Yaskawa INFORM job: OK_R2_O49(180,90)AWOK.JBI

/JOB
//NAME OK_R2_O49(180,90)AWOK
///FOLDERNAME X4
//POS
///NPOS 112,112,112,7,0,0
///TOOL 0
///POSTYPE PULSE
///PULSE
C00000=-57370,-49169,-35389,-92398,112235,2416
C00001=-57338,-39846,-12309,-87938,111954,7208
C00002=-61668,-40068,-12639,-88811,108884,7066
C00003=-63399,-40053,-12708,-89154,107656,7009
C00004=-65644,-43123,-14595,-89423,106041,7176
C00005=-66050,-42449,-14221,-89539,105759,7114
C00006=-65644,-43123,-14595,-89423,106041,7176
C00007=-63399,-40053,-12708,-89154,107656,7009
C00008=-65860,-35872,-10226,-89816,105931,6667
C00009=-67308,-37830,-11473,-89989,104891,6764
C00010=-65860,-35872,-10226,-89816,105931,6667
C00011=-63399,-40053,-12708,-89154,107656,7009
C00012=-61668,-40068,-12639,-88811,108884,7066
C00013=-57338,-39846,-12309,-87938,111954,7208
C00014=-57370,-49169,-35389,-92398,112235,2416
C00015=-56766,-48274,-34752,-92403,112675,2380
C00016=-56734,-38983,-11654,-87839,112385,7203
C00017=-61035,-39257,-12018,-88706,109335,7062
C00018=-61363,-41475,-13444,-88660,109088,7185
C00019=-65079,-42508,-14107,-89322,106443,7178
C00020=-65354,-42062,-13862,-89401,106251,7134
C00021=-65079,-42508,-14107,-89322,106443,7178
C00022=-62757,-39264,-12100,-89046,108114,7005
C00023=-65205,-35368,-10154,-89778,106406,6571
C00024=-66729,-37471,-11499,-89953,105309,6677
C00025=-65205,-35368,-10154,-89778,106406,6571
C00026=-62757,-39264,-12100,-89046,108114,7005
C00027=-61035,-39257,-12018,-88706,109335,7062
C00028=-56734,-38983,-11654,-87839,112385,7203
C00029=-56766,-48274,-34752,-92403,112675,2380
C00030=-56218,-47521,-34536,-92505,113073,2248
C00031=-56187,-38348,-11498,-87842,112791,7100
C00032=-59131,-40673,-13118,-88322,110687,7128
C00033=-64463,-43713,-15068,-89195,106879,7202
C00034=-65258,-42417,-14335,-89420,106324,7084
C00035=-65041,-42755,-14501,-89355,106475,7122
C00036=-62171,-38696,-11986,-89025,108542,6906
C00037=-64564,-34510,-9127,-89599,106856,6674
C00038=-65923,-36436,-10368,-89757,105878,6764
C00039=-64564,-34510,-9127,-89599,106856,6674
C00040=-62171,-38696,-11986,-89025,108542,6906
C00041=-60460,-38670,-11893,-88691,109758,6961
C00042=-56187,-38348,-11498,-87842,112791,7100
C00043=-58012,-44746,-32893,-92770,111760,2043
C00044=-165233,-62484,-24672,90805,98196,-8817
C00045=-158022,-60427,-23957,92500,93160,-8513
C00046=-156743,-62313,-24995,92752,92269,-8672
C00047=-155558,-59411,-23565,93051,91431,-8394
C00048=-156743,-62313,-24995,92752,92269,-8672
C00049=-159918,-59160,-23326,92117,94487,-8388
C00050=-157669,-55497,-21549,92669,92903,-8023
C00051=-156702,-56139,-21884,92856,92223,-8084
C00052=-158315,-55054,-21316,92545,93357,-7983
C00053=-165233,-62484,-24672,90805,98196,-8817
C00054=-166433,-62392,-24374,90502,99029,-8891
C00055=-159182,-60473,-23727,92230,93972,-8588
C00056=-156333,-62291,-24667,92831,91984,-8760
C00057=-155539,-60352,-23718,93033,91424,-8573
C00058=-155684,-62672,-24851,92972,91532,-8802
C00059=-160153,-59816,-23401,92033,94651,-8523
C00060=-157527,-54468,-21504,92741,92796,-7792
C00061=-156419,-55217,-21907,92950,92016,-7861
C00062=-158582,-53729,-21112,92546,93541,-7724
C00063=-166433,-62392,-24374,90502,99029,-8891
C00064=-167171,-61612,-24215,90395,99552,-8755
C00065=-159973,-59772,-23597,92089,94525,-8457
C00066=-156562,-61998,-24743,92795,92141,-8668
C00067=-155803,-60186,-23919,92988,91604,-8474
C00068=-156562,-61998,-24743,92795,92141,-8668
C00069=-161445,-58729,-23074,91799,95557,-8358
C00070=-159459,-54024,-20839,92339,94160,-7872
C00071=-157637,-55308,-21529,92681,92878,-7984
C00072=-159252,-54174,-20918,92377,94014,-7885
C00073=-167171,-61612,-24215,90395,99552,-8755
C00074=-69409,-72138,-29447,-102463,36685,-80534
C00075=-71059,-73457,-30006,-103635,35630,-80116
C00076=-71839,-65365,-14695,-121986,41568,-74598
C00077=-70275,-72833,-29744,-103069,36130,-80318
C00078=-70612,-75418,-30749,-104190,36042,-79744
C00079=-72072,-56824,-1188,-125861,43468,-72277
C00080=-72838,-56347,-1048,-126291,42972,-72187
C00081=-73459,-46502,14196,-130452,45167,-69730
C00082=-73645,-58678,-6398,-124927,41399,-73193
C00083=-74008,-49012,8836,-129230,43689,-70644
C00084=-74555,-56613,-4486,-125720,40959,-72905
C00085=-74921,-46134,12069,-130385,43538,-70149
C00086=-75408,-55045,-3275,-126310,40460,-72728
C00087=-76023,-45250,12243,-130982,42784,-70051
C00088=-76728,-63195,-18080,-121997,37141,-75456
C00089=-77109,-54539,-3849,-127025,39193,-72649
C00090=-77504,-63710,-20410,-121159,36115,-76041
C00091=-77952,-55004,-5860,-126648,38177,-73027
C00092=-56542,-67334,-11423,-115165,51876,-75640
C00093=-67053,-69065,-28106,-99490,40183,15728
C00094=-67428,-69282,-26772,-100738,40056,16409
C00095=-67529,-60027,-12907,-115722,44463,22502
C00096=-65920,-70446,-28647,-99537,41009,15920
C00097=-68407,-70268,-28636,-100327,39293,16023
C00098=-67953,-51806,517,-119653,45920,24933
C00099=-68254,-60297,-14375,-115388,43715,22147
C00100=-68715,-51405,-117,-119604,45208,24719
C00101=-69350,-59817,-14851,-115483,42822,22008
C00102=-69870,-50869,-354,-119971,44342,24699
C00103=-70281,-60433,-17733,-114511,41681,21256
C00104=-70732,-50629,-1414,-119808,43487,24415
C00105=-71119,-50129,-1155,-119967,43215,24435
C00106=-71532,-39226,16503,-124978,45598,27505
C00107=-71875,-64574,-28650,-110190,39078,18480
C00108=-72245,-56839,-15158,-115347,40339,21445
C00109=-72519,-46657,1943,-121015,42457,24796
C00110=-72775,-36077,19150,-125892,44947,27780
C00111=-71161,-41775,15932,-125497,46306,27939
BC00000=398174,725769,70942
BC00001=398174,725769,70942
BC00002=398174,725769,70942
BC00003=398174,725769,70942
BC00004=398174,725769,70942
BC00005=398174,725769,70942
BC00006=398174,725769,70942
BC00007=398174,725769,70942
BC00008=398174,725769,70942
BC00009=398174,725769,70942
BC00010=398174,725769,70942
BC00011=398174,725769,70942
BC00012=398174,725769,70942
BC00013=398174,725769,70942
BC00014=398174,725769,70942
BC00015=398174,720870,420591
BC00016=398174,720870,420591
BC00017=398174,720870,420591
BC00018=398174,720870,420591
BC00019=398174,720870,420591
BC00020=398174,720870,420591
BC00021=398174,720870,420591
BC00022=398174,720870,420591
BC00023=398174,720870,420591
BC00024=398174,720870,420591
BC00025=398174,720870,420591
BC00026=398174,720870,420591
BC00027=398174,720870,420591
BC00028=398174,720870,420591
BC00029=398174,720870,420591
BC00030=398174,716148,751922
BC00031=398174,716148,751922
BC00032=398174,716148,751922
BC00033=398174,716148,751922
BC00034=398174,716148,751922
BC00035=398174,716148,751922
BC00036=398174,716148,751922
BC00037=398174,716148,751922
BC00038=398174,716148,751922
BC00039=398174,716148,751922
BC00040=398174,716148,751922
BC00041=398174,716148,751922
BC00042=398174,716148,751922
BC00043=398174,689571,751922
BC00044=15,723854,63219
BC00045=15,723854,63219
BC00046=15,723854,63219
BC00047=15,723854,63219
BC00048=15,723854,63219
BC00049=15,723854,63219
BC00050=15,723854,63219
BC00051=15,723854,63219
BC00052=15,723854,63219
BC00053=15,723854,63219
BC00054=15,720076,395244
BC00055=15,720076,395244
BC00056=15,720076,395244
BC00057=15,720076,395244
BC00058=15,720076,395244
BC00059=15,720076,395244
BC00060=15,720076,395244
BC00061=15,720076,395244
BC00062=15,720076,395244
BC00063=15,720076,395244
BC00064=15,714414,759792
BC00065=15,714414,759792
BC00066=15,714414,759792
BC00067=15,714414,759792
BC00068=15,714414,759792
BC00069=15,714414,759792
BC00070=15,714414,759792
BC00071=15,714414,759792
BC00072=15,714414,759792
BC00073=15,714414,759792
BC00074=15,669680,870811
BC00075=15,676887,869700
BC00076=15,679769,869255
BC00077=15,679769,869255
BC00078=15,679769,869255
BC00079=15,679769,869255
BC00080=15,679769,794529
BC00081=15,679769,794529
BC00082=15,679769,652674
BC00083=15,679769,652674
BC00084=15,679769,530552
BC00085=15,679769,530552
BC00086=15,679769,409308
BC00087=15,679769,409308
BC00088=15,679769,241527
BC00089=15,679769,241527
BC00090=15,679769,105258
BC00091=15,679769,105258
BC00092=15,679769,105258
BC00093=308901,670741,873357
BC00094=311453,677596,872312
BC00095=311410,677544,872261
BC00096=312666,680852,871816
BC00097=312666,680852,871816
BC00098=311410,677544,872261
BC00099=311409,677551,750069
BC00100=311409,677551,750069
BC00101=311409,677551,629774
BC00102=311409,677551,629774
BC00103=311409,677551,498785
BC00104=311409,677551,498785
BC00105=311409,677551,426569
BC00106=311409,677551,426569
BC00107=311409,677551,187001
BC00108=311409,677551,187001
BC00109=311409,677551,187001
BC00110=311409,677551,187001
BC00111=311409,677551,187001
EC00000=1596313,556475
EC00001=1596313,556475
EC00002=1596313,556475
EC00003=1596313,556475
EC00004=1596313,556475
EC00005=1596313,556475
EC00006=1596313,556475
EC00007=1596313,556475
EC00008=1596313,556475
EC00009=1596313,556475
EC00010=1596313,556475
EC00011=1596313,556475
EC00012=1596313,556475
EC00013=1596313,556475
EC00014=1596313,556475
EC00015=1596313,556475
EC00016=1596313,556475
EC00017=1596313,556475
EC00018=1596313,556475
EC00019=1596313,556475
EC00020=1596313,556475
EC00021=1596313,556475
EC00022=1596313,556475
EC00023=1596313,556475
EC00024=1596313,556475
EC00025=1596313,556475
EC00026=1596313,556475
EC00027=1596313,556475
EC00028=1596313,556475
EC00029=1596313,556475
EC00030=1596313,556475
EC00031=1596313,556475
EC00032=1596313,556475
EC00033=1596313,556475
EC00034=1596313,556475
EC00035=1596313,556475
EC00036=1596313,556475
EC00037=1596313,556475
EC00038=1596313,556475
EC00039=1596313,556475
EC00040=1596313,556475
EC00041=1596313,556475
EC00042=1596313,556475
EC00043=1596313,556475
EC00044=1596313,556475
EC00045=1596313,556475
EC00046=1596313,556475
EC00047=1596313,556475
EC00048=1596313,556475
EC00049=1596313,556475
EC00050=1596313,556475
EC00051=1596313,556475
EC00052=1596313,556475
EC00053=1596313,556475
EC00054=1596313,556475
EC00055=1596313,556475
EC00056=1596313,556475
EC00057=1596313,556475
EC00058=1596313,556475
EC00059=1596313,556475
EC00060=1596313,556475
EC00061=1596313,556475
EC00062=1596313,556475
EC00063=1596313,556475
EC00064=1596313,556475
EC00065=1596313,556475
EC00066=1596313,556475
EC00067=1596313,556475
EC00068=1596313,556475
EC00069=1596313,556475
EC00070=1596313,556475
EC00071=1596313,556475
EC00072=1596313,556475
EC00073=1596313,556475
EC00074=1596313,556475
EC00075=1596313,556475
EC00076=1596313,556475
EC00077=1596313,556475
EC00078=1596313,556475
EC00079=1596313,556475
EC00080=1596313,556475
EC00081=1596313,556475
EC00082=1596313,556475
EC00083=1596313,556475
EC00084=1596313,556475
EC00085=1596313,556475
EC00086=1596313,556475
EC00087=1596313,556475
EC00088=1596313,556475
EC00089=1596313,556475
EC00090=1596313,556475
EC00091=1596313,556475
EC00092=1596313,556475
EC00093=1596313,556475
EC00094=1596313,556475
EC00095=1596313,556475
EC00096=1596313,556475
EC00097=1596313,556475
EC00098=1596313,556475
EC00099=1596313,556475
EC00100=1596313,556475
EC00101=1596313,556475
EC00102=1596313,556475
EC00103=1596313,556475
EC00104=1596313,556475
EC00105=1596313,556475
EC00106=1596313,556475
EC00107=1596313,556475
EC00108=1596313,556475
EC00109=1596313,556475
EC00110=1596313,556475
EC00111=1596313,556475
///POSTYPE BASE
///RECTAN
///RCONF 0,0,0,0,0,0,0,0,0,0,0,0,0,0,0,0,0,0,0,0,0,0,0,0
P00006=0.222,-3.123,-1.508,0.0000,0.0000,0.0000
P00021=-0.225,-6.128,-0.405,0.0000,0.0000,0.0000
P00022=0.222,-3.123,-1.508,0.0000,0.0000,0.0000
P00023=0.143,-0.036,0.682,0.0000,0.0000,0.0000
P00031=1.853,-0.001,-1.549,0.0000,0.0000,0.0000
P00032=1.957,0.503,-7.217,0.0000,0.0000,0.0000
///RCONF 0,0,0,0,1,0,0,0,0,0,0,0,0,0,0,0,0,0,0,0,0,0,0,0
P00033=-0.123,0.612,-5.012,0.0000,0.0000,0.0000
//INST
///DATE 2025/02/14 14:59
///ATTR SC,RW
///GROUP1 RB1,BS1
///GROUP2 ST1
NOP
'OK_r2_O49(180,90)
'Path S1126
SFTOF3D
MOVJ C00000 BC00000 VJ=100.00  +MOVJ EC00000 VJ=100.00
MOVJ C00001 BC00001 VJ=100.00  +MOVJ EC00001 VJ=100.00
MOVL C00002 BC00002 V=400.0  +MOVJ EC00002 VJ=100.00
SMOVL C00003 BC00003 V=100.0  +MOVJ EC00003
SMOVL C00004 BC00004 V=100.0  +MOVJ EC00004
SREFP 3 C00005 BC00005  +REFP EC00005
CALL JOB:SEARCH-R1-S13D
SET P031 P006
SFTON3D P031
SMOVL C00006 BC00006 V=100.0  +MOVJ EC00006
SMOVL C00007 BC00007 V=100.0  +MOVJ EC00007
SMOVL C00008 BC00008 V=100.0  +MOVJ EC00008
SREFP 3 C00009 BC00009  +REFP EC00009
CALL JOB:SEARCH-R1-S13D
SET P031 P006
SFTON3D P031
SMOVL C00010 BC00010 V=100.0  +MOVJ EC00010
SMOVL C00011 BC00011 V=100.0  +MOVJ EC00011
MOVL C00012 BC00012 V=400.0  +MOVJ EC00012 VJ=100.00
MOVL C00013 BC00013 V=1000.0  +MOVJ EC00013 VJ=100.00
MOVL C00014 BC00014 V=1000.0  +MOVJ EC00014 VJ=100.00
'Path S1127
SFTOF3D
MOVJ C00015 BC00015 VJ=100.00  +MOVJ EC00015 VJ=100.00
MOVJ C00016 BC00016 VJ=100.00  +MOVJ EC00016 VJ=100.00
MOVL C00017 BC00017 V=400.0  +MOVJ EC00017 VJ=100.00
SMOVL C00018 BC00018 V=100.0  +MOVJ EC00018
SMOVL C00019 BC00019 V=100.0  +MOVJ EC00019
SREFP 3 C00020 BC00020  +REFP EC00020
CALL JOB:SEARCH-R1-S13D
SET P032 P006
SFTON3D P032
SMOVL C00021 BC00021 V=100.0  +MOVJ EC00021
SMOVL C00022 BC00022 V=100.0  +MOVJ EC00022
SMOVL C00023 BC00023 V=100.0  +MOVJ EC00023
SREFP 3 C00024 BC00024  +REFP EC00024
CALL JOB:SEARCH-R1-S13D
SET P032 P006
SFTON3D P032
SMOVL C00025 BC00025 V=100.0  +MOVJ EC00025
SMOVL C00026 BC00026 V=100.0  +MOVJ EC00026
MOVL C00027 BC00027 V=400.0  +MOVJ EC00027 VJ=100.00
MOVL C00028 BC00028 V=1000.0  +MOVJ EC00028 VJ=100.00
MOVL C00029 BC00029 V=1000.0  +MOVJ EC00029 VJ=100.00
'Path S1128
SFTOF3D
MOVJ C00030 BC00030 VJ=100.00  +MOVJ EC00030 VJ=100.00
MOVJ C00031 BC00031 VJ=100.00  +MOVJ EC00031 VJ=100.00
MOVL C00032 BC00032 V=400.0  +MOVJ EC00032 VJ=100.00
SMOVL C00033 BC00033 V=100.0  +MOVJ EC00033
SREFP 3 C00034 BC00034  +REFP EC00034
CALL JOB:SEARCH-R1-S13D
SET P033 P006
SFTON3D P033
SMOVL C00035 BC00035 V=100.0  +MOVJ EC00035
SMOVL C00036 BC00036 V=100.0  +MOVJ EC00036
SMOVL C00037 BC00037 V=100.0  +MOVJ EC00037
SREFP 3 C00038 BC00038  +REFP EC00038
CALL JOB:SEARCH-R1-S13D
SET P033 P006
SFTON3D P033
SMOVL C00039 BC00039 V=100.0  +MOVJ EC00039
SMOVL C00040 BC00040 V=100.0  +MOVJ EC00040
MOVL C00041 BC00041 V=400.0  +MOVJ EC00041 VJ=100.00
MOVL C00042 BC00042 V=1000.0  +MOVJ EC00042 VJ=100.00
MOVL C00043 BC00043 V=1000.0  +MOVJ EC00043 VJ=100.00
'Path S1536
'DRUGA STRONA
'DRUGA STRONA
'DRUGA STRONA
SFTOF3D
MOVJ C00044 BC00044 VJ=100.00  +MOVJ EC00044 VJ=100.00
SMOVL C00045 BC00045 V=250.0  +MOVJ EC00045
SMOVL C00046 BC00046 V=100.0  +MOVJ EC00046
SREFP 3 C00047 BC00047  +REFP EC00047
CALL JOB:SEARCH-R1-S13D
SET P023 P006
SFTON3D P023
SMOVL C00048 BC00048 V=100.0  +MOVJ EC00048
SMOVL C00049 BC00049 V=100.0  +MOVJ EC00049
SMOVL C00050 BC00050 V=100.0  +MOVJ EC00050
SREFP 3 C00051 BC00051  +REFP EC00051
CALL JOB:SEARCH-R1-S13D
SET P023 P006
SFTON3D P023
SMOVL C00052 BC00052 V=100.0  +MOVJ EC00052
MOVL C00053 BC00053 V=1000.0  +MOVJ EC00053 VJ=100.00
'Path S1537
SFTOF3D
MOVJ C00054 BC00054 VJ=100.00  +MOVJ EC00054 VJ=100.00
SMOVL C00055 BC00055 V=250.0  +MOVJ EC00055
SMOVL C00056 BC00056 V=100.0  +MOVJ EC00056
SREFP 3 C00057 BC00057  +REFP EC00057
CALL JOB:SEARCH-R1-S13D
SET P022 P006
SFTON3D P022
SMOVL C00058 BC00058 V=100.0  +MOVJ EC00058
SMOVL C00059 BC00059 V=166.7  +MOVJ EC00059
SMOVL C00060 BC00060 V=100.0  +MOVJ EC00060
SREFP 3 C00061 BC00061  +REFP EC00061
CALL JOB:SEARCH-R1-S13D
SET P022 P006
SFTON3D P022
SMOVL C00062 BC00062 V=100.0  +MOVJ EC00062
MOVL C00063 BC00063 V=1000.0  +MOVJ EC00063 VJ=100.00
'Path S1538
SFTOF3D
MOVJ C00064 BC00064 VJ=100.00  +MOVJ EC00064 VJ=100.00
SMOVL C00065 BC00065 V=333.3  +MOVJ EC00065
SMOVL C00066 BC00066 V=100.0  +MOVJ EC00066
SREFP 3 C00067 BC00067  +REFP EC00067
CALL JOB:SEARCH-R1-S13D
SET P021 P006
SFTON3D P021
SMOVL C00068 BC00068 V=100.0  +MOVJ EC00068
SMOVL C00069 BC00069 V=166.7  +MOVJ EC00069
SMOVL C00070 BC00070 V=100.0  +MOVJ EC00070
SREFP 3 C00071 BC00071  +REFP EC00071
CALL JOB:SEARCH-R1-S13D
SET P021 P006
SFTON3D P021
SMOVL C00072 BC00072 V=100.0  +MOVJ EC00072
MOVL C00073 BC00073 V=1000.0  +MOVJ EC00073 VJ=100.00
'Path W1539
SFTOF3D
SFTON3D P021
MOVJ C00074 BC00074 VJ=100.00  +MOVJ EC00074 VJ=100.00
SMOVL C00075 BC00075 V=166.7  +MOVJ EC00075
SMOVL C00076 BC00076 V=133.3 PL=0  +MOVJ EC00076
SREFP 1 C00077 BC00077  +REFP EC00077
SREFP 2 C00078 BC00078  +REFP EC00078
MACRO1 MJ#(0) ARGF6
ARCON
SFTON3D P021
SMOVL C00079 BC00079 V=10.0  +MOVJ EC00079
ARCOF
SMOVL C00080 BC00080 V=500.0  +MOVJ EC00080
ARCON
SMOVL C00081 BC00081 V=10.0  +MOVJ EC00081
ARCOF
SFTON3D P022
SMOVL C00082 BC00082 V=500.0  +MOVJ EC00082
ARCON
SMOVL C00083 BC00083 V=10.0  +MOVJ EC00083
ARCOF
SMOVL C00084 BC00084 V=500.0  +MOVJ EC00084
ARCON
SMOVL C00085 BC00085 V=10.0  +MOVJ EC00085
ARCOF
SMOVL C00086 BC00086 V=500.0  +MOVJ EC00086
ARCON
SMOVL C00087 BC00087 V=10.0  +MOVJ EC00087
ARCOF
SFTON3D P023
SMOVL C00088 BC00088 V=500.0  +MOVJ EC00088
ARCON
SMOVL C00089 BC00089 V=10.0  +MOVJ EC00089
ARCOF
SMOVL C00090 BC00090 V=500.0  +MOVJ EC00090
ARCON
SMOVL C00091 BC00091 V=10.0  +MOVJ EC00091
ARCOF
SFTOF3D
MOVJ C00092 BC00092 VJ=100.00  +MOVJ EC00092 VJ=100.00
SFTOF3D
'Path W343
SFTOF3D
MOVJ C00093 BC00093 VJ=100.00  +MOVJ EC00093 VJ=100.00
SMOVL C00094 BC00094 V=400.0  +MOVJ EC00094
SFTON3D P033
SMOVL C00095 BC00095 V=133.3 PL=0  +MOVJ EC00095
SREFP 1 C00096 BC00096  +REFP EC00096
SREFP 2 C00097 BC00097  +REFP EC00097
MACRO1 MJ#(0) ARGF6
ARCON
SMOVL C00098 BC00098 V=10.0  +MOVJ EC00098
ARCOF
SMOVL C00099 BC00099 V=166.7  +MOVJ EC00099
ARCON
SMOVL C00100 BC00100 V=10.0  +MOVJ EC00100
ARCOF
SFTON3D P032
SMOVL C00101 BC00101 V=500.0  +MOVJ EC00101
ARCON
SMOVL C00102 BC00102 V=10.0  +MOVJ EC00102
ARCOF
SMOVL C00103 BC00103 V=500.0  +MOVJ EC00103
ARCON
SMOVL C00104 BC00104 V=10.0  +MOVJ EC00104
ARCOF
SFTON3D P031
SMOVL C00105 BC00105 V=500.0  +MOVJ EC00105
ARCON
SMOVL C00106 BC00106 V=10.0  +MOVJ EC00106
ARCOF
SFTON3D P031
SMOVL C00107 BC00107 V=500.0  +MOVJ EC00107
ARCON
SMOVL C00108 BC00108 V=10.0  +MOVJ EC00108
ARCOF
SMOVL C00109 BC00109 V=500.0  +MOVJ EC00109
ARCON
SMOVL C00110 BC00110 V=10.0  +MOVJ EC00110
ARCOF
SMOVL C00111 BC00111 V=1000.0  +MOVJ EC00111
SFTOF3D
END
